(* PLC project Trafic_Light, Unknown Unnamed 1 *)
(* stored: creationDateTime 2020-10-12T21:33:17, modificationDateTime 2020-10-13T22:32:39 *)

PROGRAM Trafic_light
  VAR
    TOF0 : TOF;
    Always_True : BOOL := True;  (* Always True - Do not force off *)
    Delay_PLC_start_up : BOOL;  (* Made to make sure no false negative flanks are picked up by the PLC program *)
    TOF1 : TOF;
    TOF2 : TOF;
  END_VAR
  VAR
    O_LEDRed AT %QX100.0 : BOOL;  (* This can be a red LED on pin 7 *)
    O_LEDOrange AT %QX100.1 : BOOL;  (* This can be a orange LED on pin 8 *)
    O_LEDGreen AT %QX100.2 : BOOL;  (* This can be a Green LED on pin 12 *)
  END_VAR
  VAR
    No_lamps_active_for_1s : BOOL;
    F_TRIG0 : F_TRIG;
    F_TRIG1 : F_TRIG;
    F_TRIG2 : F_TRIG;
    TON0 : TON;
    SR0 : SR;
    TOF3 : TOF;
    TOF4 : TOF;
    TOF5 : TOF;
  END_VAR

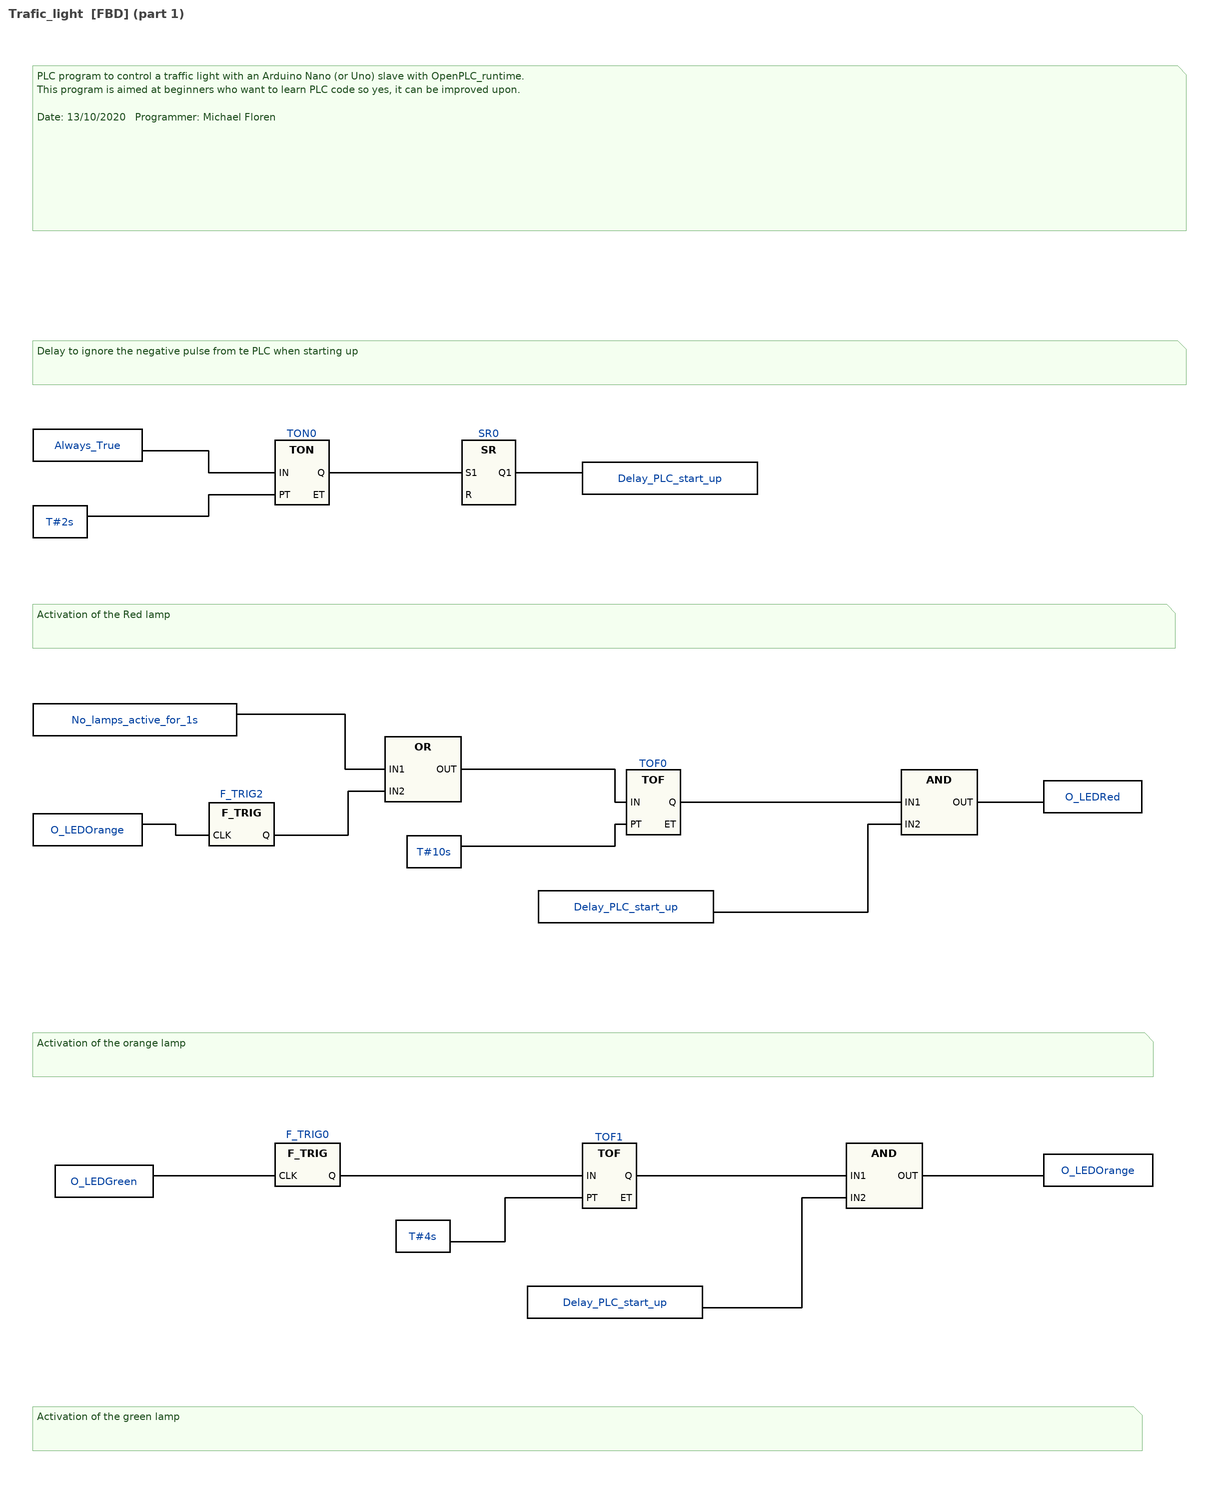
(* FBD diagram, written out as Structured Text *)
(* PLC program to control a traffic light with an Arduino Nano (or Uno) slave with OpenPLC_runtime. 
This program is aimed at beginners who want to learn PLC code so yes, it can be improved upon. 

Date: 13/10/2020   Programmer: Michael Floren *)
(* Delay to ignore the negative pulse from te PLC when starting up *)
TON0(IN := Always_True, PT := T#2s);
SR0(S1 := TON0.Q);
Delay_PLC_start_up := SR0.Q1;
(* Activation of the Red lamp *)
F_TRIG2(CLK := O_LEDOrange);
TOF0(IN := No_lamps_active_for_1s OR F_TRIG2.Q, PT := T#10s);
O_LEDRed := TOF0.Q AND Delay_PLC_start_up;
(* Activation of the orange lamp *)
F_TRIG0(CLK := O_LEDGreen);
TOF1(IN := F_TRIG0.Q, PT := T#4s);
O_LEDOrange := TOF1.Q AND Delay_PLC_start_up;
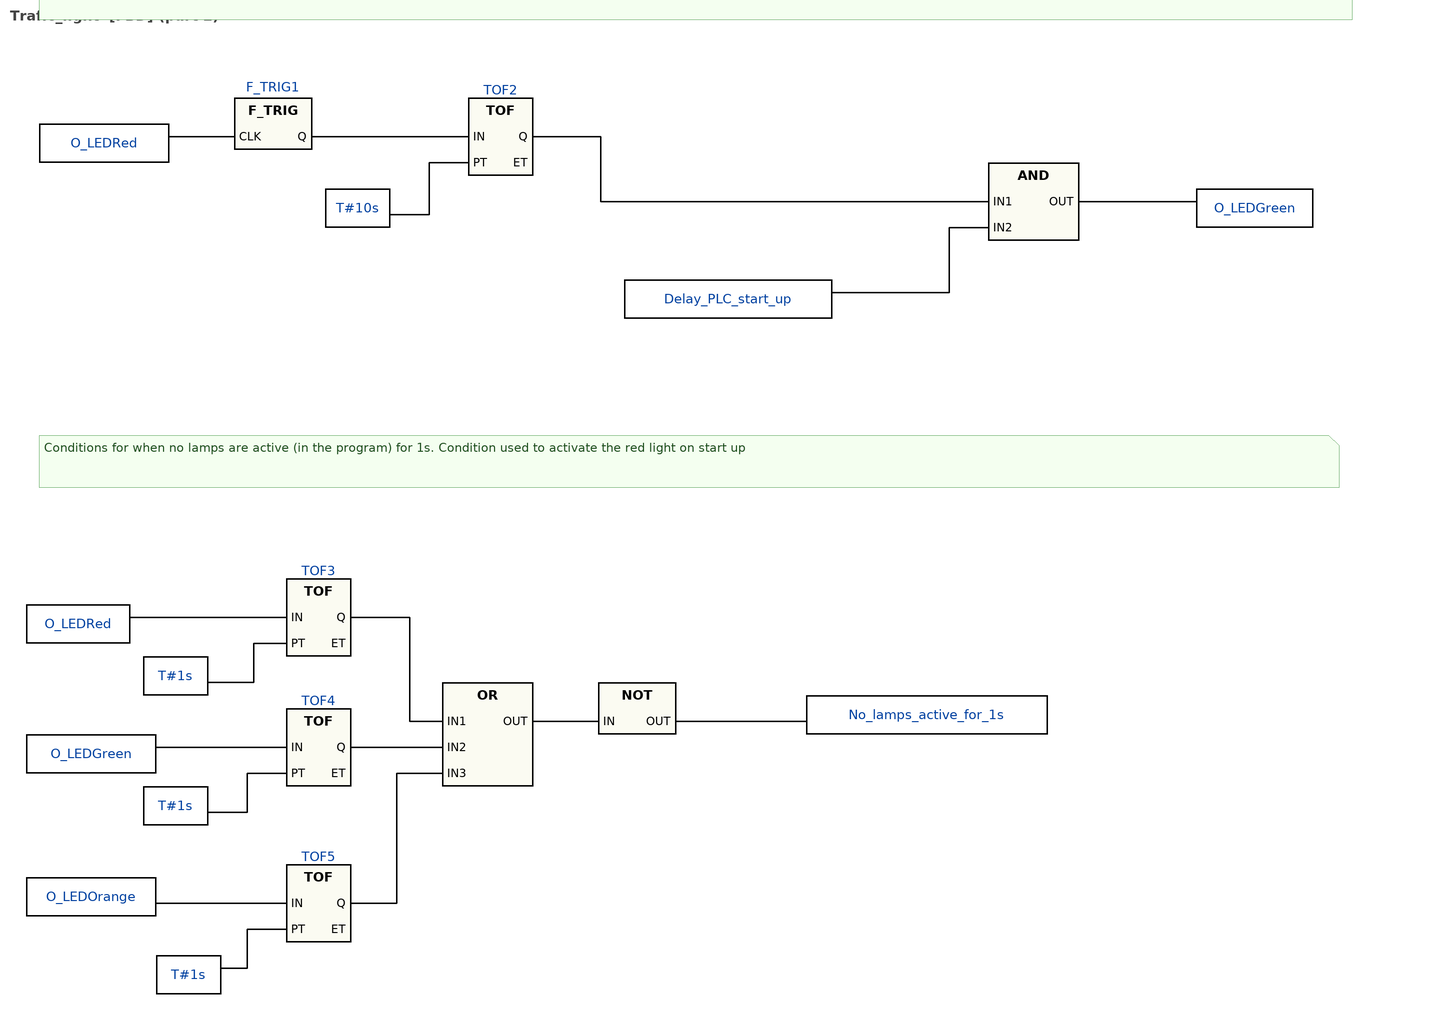
(* Activation of the green lamp *)
F_TRIG1(CLK := O_LEDRed);
TOF2(IN := F_TRIG1.Q, PT := T#10s);
O_LEDGreen := TOF2.Q AND Delay_PLC_start_up;
(* Conditions for when no lamps are active (in the program) for 1s. Condition used to activate the red light on start up *)
TOF3(IN := O_LEDRed, PT := T#1s);
TOF4(IN := O_LEDGreen, PT := T#1s);
TOF5(IN := O_LEDOrange, PT := T#1s);
No_lamps_active_for_1s := NOT (TOF3.Q OR TOF4.Q OR TOF5.Q);
END_PROGRAM

CONFIGURATION Config0
  RESOURCE Res0 ON PLC
    TASK task0(INTERVAL := T#20ms, PRIORITY := 0);
    PROGRAM instance0 WITH task0 : Trafic_light;
  END_RESOURCE
END_CONFIGURATION
